// TIA Portal project "PLC Toggle Output with Pushbutton" (V17)
// Pushbutton ON/OFF
// When pushbutton is pressed and released, then the output will be ON.
// When pushbutton is again pressed and released, then the output will be OFF.

(* hardware
DEVICE "S7-1200 station_1"  S7-1200 Station
   slot 0: "Rack_0"  S7-1200 Rack  Rack  V1.0
   slot 1: "PLC_1"  CPU 1212C AC/DC/Rly  6ES7 212-1BE40-0XB0  V4.5
*)

// ===== PLC "PLC_1"  CPU 1212C AC/DC/Rly =====

VAR_GLOBAL   // PLC tag table "Default tag table"
   "PB" AT %I0.0 : Bool;
   "Motor" AT %Q0.0 : Bool;
   "Tag_1" AT %M0.0 : Bool;
   "Tag_2" AT %M0.1 : Bool;
END_VAR

ORGANIZATION_BLOCK "Main"   // OB1, LAD, ProgramCycle
TITLE = "Main Program Sweep (Cycle)"
{ S7_Optimized_Access := 'TRUE' }
VERSION : 0.1
   VAR_INPUT
      Initial_Call : Bool;   // Initial call of this OB
      Remanence : Bool;   // =True, if remanent data are available
   END_VAR
BEGIN

REGION Network 1
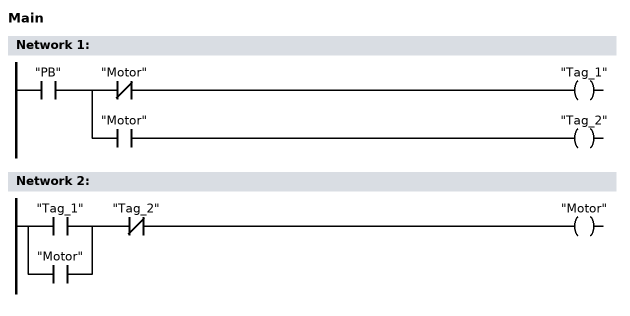
   RUNG wire#powerrail
      Contact( "PB" )
      wire#w1
      I_Contact( "Motor" )
      Coil( "Tag_1" )
   END_RUNG
   RUNG wire#w1
      Contact( "Motor" )
      Coil( "Tag_2" )
   END_RUNG
   // the same network as SCL:
   "Tag_1" := "PB" AND NOT "Motor";
   "Tag_2" := "PB" AND "Motor";
END_REGION

REGION Network 2
   RUNG wire#powerrail
      Contact( "Tag_1" )
      wire#w1
      I_Contact( "Tag_2" )
      Coil( "Motor" )
   END_RUNG
   RUNG wire#powerrail
      Contact( "Motor" )
   END_RUNG wire#w1
   // the same network as SCL:
   "Motor" := ("Tag_1" OR "Motor") AND NOT "Tag_2";
END_REGION
END_ORGANIZATION_BLOCK